(* IEC 61131-3 sources: WATT_Offline/HTB/Prolabs/Alchemy/1. 10.10.110.21/Git, 6 files *)

(* ---- bottle_filling.st ---- *)
PROGRAM botte_filling
  VAR_INPUT
    start : BOOL;
    stop : BOOL;
    overflow_sensor : BOOL;
    filling_sensor : BOOL;
    level_sensor : BOOL;
    capping_sensor : BOOL;
    cap_lazer_sensor : BOOL;
    empty_tank_sensor : BOOL;
  END_VAR
  VAR_OUTPUT
    process_start : BOOL;
    solenoid_valve : BOOL;
    motor_cap : BOOL;
    conveyor_motor : BOOL;
  END_VAR
  VAR
    batch_completed : BOOL;
    sp_beer_flow : INT;
    batch_no : INT;
    current_batch : INT;
    CTU0 : CTU;
    R_TRIG1 : R_TRIG;
  END_VAR

  process_start := NOT(empty_tank_sensor) AND NOT(overflow_sensor) AND NOT(stop) AND (process_start OR start);

  // Hardcoded value min:0 max:100
  sp_beer_flow := 5;

  conveyor_motor := (NOT(motor_cap) OR NOT(capping_sensor)) AND process_start AND (NOT(solenoid_valve) OR NOT(filling_sensor));
  solenoid_valve := NOT(level_sensor) AND (filling_sensor OR solenoid_valve) AND process_start;
  motor_cap := NOT(cap_lazer_sensor) AND (capping_sensor OR motor_cap) AND process_start;
  R_TRIG1(CLK := motor_cap);
  CTU0(CU := R_TRIG1.Q, R := NOT(process_start), PV := batch_no);
  batch_completed := CTU0.Q;
  current_batch := CTU0.CV;
END_PROGRAM

CONFIGURATION Config0

  RESOURCE Res0 ON PLC
    TASK task0(INTERVAL := T#10ms,PRIORITY := 0);
    PROGRAM instance0 WITH task0 : botte_filling;
  END_RESOURCE
END_CONFIGURATION

(* ---- conditioning_aging.st ---- *)
PROGRAM pressure_control
  VAR_EXTERNAL
    master : BOOL;
  END_VAR
  VAR_INPUT
    pressure_sensor : INT := 10;
  END_VAR
  VAR_OUTPUT
    sp_pressure : INT;
    pressure_valve : BOOL;
    open_pressure_valve : BOOL;
    close_pressure_valve : BOOL;
  END_VAR
  VAR
    _TMP_ADD52_OUT : INT;
    _TMP_GT14_OUT : BOOL;
    _TMP_SUB48_OUT : INT;
    _TMP_LT51_OUT : BOOL;
  END_VAR

  pressure_valve := NOT(close_pressure_valve) AND open_pressure_valve AND master;
  _TMP_ADD52_OUT := ADD(sp_pressure, 2);
  _TMP_GT14_OUT := GT(pressure_sensor, _TMP_ADD52_OUT);
  open_pressure_valve := master AND _TMP_GT14_OUT;
  _TMP_SUB48_OUT := SUB(sp_pressure, 2);
  _TMP_LT51_OUT := LT(pressure_sensor, _TMP_SUB48_OUT);
  close_pressure_valve := master AND _TMP_LT51_OUT;
END_PROGRAM

PROGRAM temperature_control
  VAR_EXTERNAL
    master : BOOL;
  END_VAR
  VAR_INPUT
    temp : INT;
  END_VAR
  VAR_OUTPUT
    heater : BOOL;
    sp_heater : INT;
    heater_start : BOOL;
    heater_stop : BOOL;
    cooler : BOOL;
    sp_cooler : INT;
    cooler_start : BOOL;
    cooler_stop : BOOL;
  END_VAR
  VAR
    _TMP_SUB48_OUT : INT;
    _TMP_LT51_OUT : BOOL;
    _TMP_ADD52_OUT : INT;
    _TMP_GT14_OUT : BOOL;
    _TMP_ADD45_OUT : INT;
    _TMP_GT9_OUT : BOOL;
    _TMP_SUB41_OUT : INT;
    _TMP_LT44_OUT : BOOL;
  END_VAR

  heater := NOT(heater_stop) AND (heater OR heater_start) AND master;
  _TMP_SUB48_OUT := SUB(sp_heater, 2);
  _TMP_LT51_OUT := LT(temp, _TMP_SUB48_OUT);
  heater_start := master AND _TMP_LT51_OUT;
  _TMP_ADD52_OUT := ADD(sp_heater, 2);
  _TMP_GT14_OUT := GT(temp, _TMP_ADD52_OUT);
  heater_stop := master AND _TMP_GT14_OUT;
  cooler := NOT(cooler_stop) AND (cooler OR cooler_start) AND master;
  _TMP_ADD45_OUT := ADD(sp_cooler, 2);
  _TMP_GT9_OUT := GT(temp, _TMP_ADD45_OUT);
  cooler_start := master AND _TMP_GT9_OUT;
  _TMP_SUB41_OUT := SUB(sp_cooler, 2);
  _TMP_LT44_OUT := LT(temp, _TMP_SUB41_OUT);
  cooler_stop := master AND _TMP_LT44_OUT;
END_PROGRAM

PROGRAM conditioning
  VAR_EXTERNAL
    master : BOOL;
  END_VAR
  VAR_INPUT
    start : BOOL;
    stop : BOOL;
    open_output_valve : BOOL;
    ultrasonic_level : INT;
  END_VAR
  VAR_OUTPUT
    cycle_on : BOOL;
    intake_pump_material_a : BOOL;
    stop_intake_a : BOOL;
    output_valve : BOOL;
    conditioning_completed : BOOL;
    sp_conditioning_time : INT;
    sp_material_a : INT;
    elapsed_time : INT;
    conditioing_time : TIME;
    elapsed_time_t : TIME;
  END_VAR
  VAR
    TON0 : TON;
    _TMP_GE15_OUT : BOOL;
    _TMP_INT_TO_TIME67_OUT : TIME;
    _TMP_TIME_TO_INT68_OUT : INT;
  END_VAR

  cycle_on := NOT(stop) AND (cycle_on OR start);
  master := NOT(stop) AND (cycle_on OR start);
  intake_pump_material_a := NOT(stop_intake_a) AND cycle_on;
  _TMP_GE15_OUT := GE(ultrasonic_level, sp_material_a);
  stop_intake_a := cycle_on AND _TMP_GE15_OUT;
  _TMP_INT_TO_TIME67_OUT := INT_TO_TIME(sp_conditioning_time);
  conditioing_time := _TMP_INT_TO_TIME67_OUT;
  TON0(IN := stop_intake_a AND cycle_on, PT := conditioing_time);
  conditioning_completed := TON0.Q;
  elapsed_time_t := TON0.ET;
  _TMP_TIME_TO_INT68_OUT := TIME_TO_INT(elapsed_time_t);
  elapsed_time := _TMP_TIME_TO_INT68_OUT;
  output_valve := open_output_valve AND conditioning_completed AND cycle_on;
END_PROGRAM

CONFIGURATION Config0

  RESOURCE Res0 ON PLC
    VAR_GLOBAL
      master : BOOL;
    END_VAR
    TASK task0(INTERVAL := T#1s0ms,PRIORITY := 0);
    TASK task1(INTERVAL := T#1s0ms,PRIORITY := 0);
    TASK task2(INTERVAL := T#1s0ms,PRIORITY := 0);
    PROGRAM instance0 WITH task0 : conditioning;
    PROGRAM instance2 WITH task0 : pressure_control;
    PROGRAM instance1 WITH task1 : temperature_control;
  END_RESOURCE
END_CONFIGURATION

(* ---- fermentation.st ---- *)
PROGRAM fermentation
  VAR_OUTPUT
    sp201 : INT;
    sp202 : INT;
    sp203 : INT;
    sp204 : INT;
  END_VAR
  VAR_EXTERNAL
    MASTER : BOOL;
  END_VAR
  VAR_INPUT
    Start : BOOL;
    Stop : BOOL;
    ultrasonic_level : INT;
  END_VAR
  VAR_OUTPUT
    cycle_on : BOOL;
    intake_pump_material_a : BOOL;
    intake_pump_material_b : BOOL;
    stop_intake_a : BOOL;
    stop_intake_b : BOOL;
    allow_intake_b : BOOL;
    agitator_motor : BOOL;
    stage_timer : BOOL;
    stage_completed : BOOL;
    stage_time : TIME;
    elapsed_stage_timer : TIME;
    elapsed_stage_time : INT;
    sp_agitator_speed : INT;
    next_stage : BOOL;
  END_VAR
  VAR_INPUT
    temp_sensor : INT;
  END_VAR
  VAR_OUTPUT
    stop_agitation : BOOL;
  END_VAR
  VAR
    TON1 : TON;
    _TMP_GE15_OUT : BOOL;
    _TMP_GE9_OUT : BOOL;
    _TMP_GE77_OUT : BOOL;
    _TMP_INT_TO_TIME72_OUT : TIME;
    _TMP_TIME_TO_INT79_OUT : INT;
  END_VAR

  cycle_on := NOT(Stop) AND (Start OR cycle_on);
  MASTER := NOT(Stop) AND (Start OR cycle_on);

  intake_pump_material_a := NOT(stop_intake_a) AND cycle_on;

  _TMP_GE15_OUT := GE(ultrasonic_level, sp201);
  stop_intake_a := cycle_on AND _TMP_GE15_OUT;

  intake_pump_material_b := NOT(stop_intake_b) AND (allow_intake_b OR intake_pump_material_b) AND

  stop_intake_a AND cycle_on;

  _TMP_GE9_OUT := GE(temp_sensor, sp203);
  allow_intake_b := _TMP_GE9_OUT;

  _TMP_GE77_OUT := GE(ultrasonic_level, sp202);
  stop_intake_b := cycle_on AND _TMP_GE77_OUT;

  _TMP_INT_TO_TIME_MIN72_OUT := INT_TO_TIME_MIN(sp204);
  stage_time := _TMP_INT_TO_TIME_MIN72_OUT;

  agitator_motor := NOT(stop_agitation) AND (agitator_motor OR stop_intake_a) AND cycle_on;

  TON1(IN := next_stage AND cycle_on, PT := stage_time);
  stage_timer := TON1.Q;
  elapsed_stage_timer := TON1.ET;

  _TMP_TIME_TO_INT79_OUT := TIME_TO_INT(elapsed_stage_timer);
  elapsed_stage_time := _TMP_TIME_TO_INT79_OUT;

  stage_completed := stage_timer AND cycle_on;
END_PROGRAM

PROGRAM pressure_control
  VAR_EXTERNAL
    MASTER : BOOL;
  END_VAR
  VAR_OUTPUT
    sp208 : INT;
    sp209 : INT;
  END_VAR
  VAR_INPUT
    pressure_sensor : INT;
  END_VAR
  VAR_OUTPUT
    pressure_valve : BOOL;
    open_pressure_valve : BOOL;
    close_pressure_valve : BOOL;
  END_VAR
  VAR
    _TMP_ADD52_OUT : INT;
    _TMP_GT14_OUT : BOOL;
    _TMP_SUB48_OUT : INT;
    _TMP_LT51_OUT : BOOL;
  END_VAR

  pressure_valve := NOT(close_pressure_valve) AND open_pressure_valve AND MASTER;
  _TMP_ADD52_OUT := ADD(sp208, sp209);
  _TMP_GT14_OUT := GT(pressure_sensor, _TMP_ADD52_OUT);
  open_pressure_valve := MASTER AND _TMP_GT14_OUT;
  _TMP_SUB48_OUT := SUB(sp208, sp209);
  _TMP_LT51_OUT := LT(pressure_sensor, _TMP_SUB48_OUT);
  close_pressure_valve := MASTER AND _TMP_LT51_OUT;
END_PROGRAM

PROGRAM pH_control
  VAR_EXTERNAL
    MASTER : BOOL;
  END_VAR
  VAR_OUTPUT
    sp210 : INT;
    sp211 : INT;
    sp212 : INT;
    active : BOOL;
    base_pump : BOOL;
    base_start : BOOL;
    base_stop : BOOL;
    acid_pump : BOOL;
    acid_start : BOOL;
    acid_stop : BOOL;
  END_VAR
  VAR_INPUT
    ph_sensor : INT;
  END_VAR
  VAR
    _TMP_SUB48_OUT : INT;
    _TMP_LT51_OUT : BOOL;
    _TMP_ADD45_OUT : INT;
    _TMP_GT9_OUT : BOOL;
    _TMP_ADD52_OUT : INT;
    _TMP_GT14_OUT : BOOL;
    _TMP_SUB41_OUT : INT;
    _TMP_LT44_OUT : BOOL;
  END_VAR

  base_pump := NOT(base_stop) AND (base_pump OR base_start) AND MASTER;
  acid_pump := NOT(acid_stop) AND (acid_pump OR acid_start) AND MASTER;

  _TMP_SUB48_OUT := SUB(sp210, sp211);
  _TMP_LT51_OUT := LT(ph_sensor, _TMP_SUB48_OUT);
  base_start := MASTER AND _TMP_LT51_OUT;

  _TMP_ADD45_OUT := ADD(sp210, sp212);
  _TMP_GT9_OUT := GT(ph_sensor, _TMP_ADD45_OUT);
  acid_start := MASTER AND _TMP_GT9_OUT;

  _TMP_ADD52_OUT := ADD(sp210, sp211);
  _TMP_GT14_OUT := GT(ph_sensor, _TMP_ADD52_OUT);
  base_stop := MASTER AND _TMP_GT14_OUT;

  _TMP_SUB41_OUT := SUB(sp210, sp212);
  _TMP_LT44_OUT := LT(ph_sensor, _TMP_SUB41_OUT);
  acid_stop := MASTER AND _TMP_LT44_OUT;
END_PROGRAM

PROGRAM temperature_control
  VAR_EXTERNAL
    MASTER : BOOL;
  END_VAR
  VAR_OUTPUT
    sp205 : INT;
    sp206 : INT;
    sp207 : INT;
  END_VAR
  VAR_INPUT
    temp_sensor : INT;
  END_VAR
  VAR_OUTPUT
    heater : BOOL;
    heater_start : BOOL;
    heater_stop : BOOL;
    cooler : BOOL;
    cooler_start : BOOL;
    cooler_stop : BOOL;
  END_VAR
  VAR
    _TMP_SUB48_OUT : INT;
    _TMP_LT51_OUT : BOOL;
    _TMP_ADD45_OUT : INT;
    _TMP_GT9_OUT : BOOL;
    _TMP_ADD52_OUT : INT;
    _TMP_GT14_OUT : BOOL;
    _TMP_SUB41_OUT : INT;
    _TMP_LT44_OUT : BOOL;
  END_VAR

  heater := NOT(heater_stop) AND (heater OR heater_start) AND MASTER;
  cooler := NOT(cooler_stop) AND (cooler OR cooler_start) AND MASTER;

  _TMP_SUB48_OUT := SUB(sp205, sp207);
  _TMP_LT51_OUT := LT(temp_sensor, _TMP_SUB48_OUT);
  heater_start := MASTER AND _TMP_LT51_OUT;

  _TMP_ADD45_OUT := ADD(sp206, sp207);
  _TMP_GT9_OUT := GT(temp_sensor, _TMP_ADD45_OUT);
  cooler_start := MASTER AND _TMP_GT9_OUT;

  _TMP_ADD52_OUT := ADD(sp205, sp207);
  _TMP_GT14_OUT := GT(temp_sensor, _TMP_ADD52_OUT);
  heater_stop := MASTER AND _TMP_GT14_OUT;

  _TMP_SUB41_OUT := SUB(sp206, sp207);
  _TMP_LT44_OUT := LT(temp_sensor, _TMP_SUB41_OUT);
  cooler_stop := MASTER AND _TMP_LT44_OUT;
END_PROGRAM

PROGRAM od_control
  VAR_EXTERNAL
    MASTER : BOOL;
  END_VAR
  VAR_OUTPUT
    sp213 : INT;
    sp214 : INT;
  END_VAR
  VAR_INPUT
    do_sensor : INT;
  END_VAR
  VAR_OUTPUT
    aeration_valve : BOOL;
    open_valve : BOOL;
    close_valve : BOOL;
  END_VAR
  VAR
    _TMP_SUB48_OUT : INT;
    _TMP_LT51_OUT : BOOL;
    _TMP_ADD52_OUT : INT;
    _TMP_GE53_OUT : BOOL;
  END_VAR

  aeration_valve := NOT(close_valve) AND (aeration_valve OR open_valve) AND MASTER;

  _TMP_SUB48_OUT := SUB(sp213, sp214);
  _TMP_LT51_OUT := LT(do_sensor, _TMP_SUB48_OUT);
  open_valve := MASTER AND _TMP_LT51_OUT;

  _TMP_ADD52_OUT := ADD(sp213, sp214);
  _TMP_GE53_OUT := GE(do_sensor, _TMP_ADD52_OUT);
  close_valve := MASTER AND _TMP_GE53_OUT;
END_PROGRAM

CONFIGURATION Config0

  RESOURCE Res0 ON PLC
    VAR_GLOBAL
      MASTER : BOOL;
    END_VAR
    TASK task0(INTERVAL := T#20ms,PRIORITY := 0);
    TASK task1(INTERVAL := T#20ms,PRIORITY := 0);
    TASK task2(INTERVAL := T#20ms,PRIORITY := 0);
    TASK task3(INTERVAL := T#20ms,PRIORITY := 0);
    TASK task4(INTERVAL := T#20ms,PRIORITY := 0);
    PROGRAM instance0 WITH task0 : fermentation;
    PROGRAM instance2 WITH task0 : pressure_control;
    PROGRAM instance4 WITH task0 : od_control;
    PROGRAM instance1 WITH task1 : temperature_control;
    PROGRAM instance3 WITH task3 : pH_control;
  END_RESOURCE
END_CONFIGURATION

(* ---- lautering.st ---- *)
PROGRAM lauter_tun
  VAR_INPUT
    start : BOOL;
    stop : BOOL;
    turbidity_sensor : INT;
    ultra_level_sensor : INT;
  END_VAR
  VAR_OUTPUT
    process_start : BOOL;
    output_valve : BOOL;
    intake_a : BOOL;
    sparge_water_valve : BOOL;
    stop_intake_a : BOOL;
    stop_sparge_water : BOOL;
    rake : BOOL;
    recirculation_pump : BOOL;
    rake_stop : BOOL;
    r_pump_stop : BOOL;
    settling_completed : BOOL;
    grain_removal : BOOL;
    stop_first_runoff : BOOL;
    stop_removal : BOOL;
    stop_final_runoff : BOOL;
    sp_mash_lvl AT %MW10 : INT;
    sp_sparge_water_temp AT %MW11 : INT;
    sp_settle_phase AT %MW51 : INT;
    sp_sparge_water_lvl AT %MW52 : INT;
    sp_first_runoff AT %MW44 : INT;
    sp_grain_bed_level AT %MW35 : INT;
    sp_turbidity_rake AT %MW23 : INT;
    sp_turbidity_vor AT %MW22 : INT;
  END_VAR
  VAR
    settle_phase_pt : TIME;
    settle_phase_et : TIME;
    sp_rake_timer : TIME;
    TON1 : TON;
    TON0 : TON;
    _TMP_GE28_OUT : BOOL;
    _TMP_INT_TO_TIME91_OUT : TIME;
    _TMP_LT62_OUT : BOOL;
    _TMP_LE89_OUT : BOOL;
    _TMP_LE102_OUT : BOOL;
    _TMP_GE107_OUT : BOOL;
    _TMP_LT123_OUT : BOOL;
    _TMP_LT114_OUT : BOOL;
  END_VAR

  process_start := NOT(stop) AND start;
  intake_a := NOT(stop_intake_a) AND process_start;
  _TMP_GE28_OUT := GE(ultra_level_sensor, sp_mash_lvl);
  stop_intake_a := process_start AND _TMP_GE28_OUT OR stop_intake_a AND process_start;
  _TMP_INT_TO_TIME91_OUT := INT_TO_TIME(sp_settle_phase);
  settle_phase_pt := _TMP_INT_TO_TIME91_OUT;
  TON0(IN := stop_intake_a AND process_start, PT := settle_phase_pt);
  settling_completed := TON0.Q;
  settle_phase_et := TON0.ET;
  rake := NOT(rake_stop) AND (rake OR settling_completed) AND process_start;
  _TMP_LT62_OUT := LT(turbidity_sensor, sp_turbidity_rake);
  TON1(IN := stop_intake_a AND process_start AND _TMP_LT62_OUT, PT := sp_rake_timer);
  rake_stop := TON1.Q;
  recirculation_pump := NOT(r_pump_stop) AND (recirculation_pump OR settling_completed) AND process_start;
  _TMP_LE89_OUT := LE(turbidity_sensor, sp_turbidity_vor);
  r_pump_stop := rake_stop AND process_start AND _TMP_LE89_OUT;
  output_valve := NOT(stop_first_runoff) AND (output_valve OR r_pump_stop) AND process_start;
  _TMP_LE102_OUT := LE(ultra_level_sensor, sp_first_runoff);
  stop_first_runoff := r_pump_stop AND process_start AND _TMP_LE102_OUT OR stop_first_runoff AND process_start;
  sparge_water_valve := NOT(stop_sparge_water) AND stop_first_runoff AND process_start;
  _TMP_GE107_OUT := GE(ultra_level_sensor, sp_sparge_water_lvl);
  stop_sparge_water := stop_first_runoff AND process_start AND _TMP_GE107_OUT OR stop_sparge_water;
  output_valve := NOT(stop_final_runoff) AND (output_valve OR stop_sparge_water) AND process_start;
  _TMP_LT123_OUT := LT(ultra_level_sensor, sp_grain_bed_level);
  stop_final_runoff := stop_sparge_water AND process_start AND _TMP_LT123_OUT;
  grain_removal := NOT(stop_removal) AND (grain_removal OR stop_final_runoff) AND process_start;
  _TMP_LT114_OUT := LT(ultra_level_sensor, 5);
  stop_removal := stop_final_runoff AND process_start AND _TMP_LT114_OUT;
END_PROGRAM

CONFIGURATION Config0

  RESOURCE Res0 ON PLC
    TASK task0(INTERVAL := T#1s0ms,PRIORITY := 0);
    PROGRAM instance0 WITH task0 : lauter_tun;
  END_RESOURCE
END_CONFIGURATION

(* ---- mash_mixing.st ---- *)
PROGRAM pressure_control
  VAR_EXTERNAL
    MASTER : BOOL;
  END_VAR
  VAR_INPUT
    pressure_sensor : INT;
  END_VAR
  VAR_OUTPUT
    sp_pressure : INT;
    pressure_valve : BOOL;
    open_pressure_valve : BOOL;
    close_pressure_valve : BOOL;
  END_VAR
  VAR
    _TMP_ADD52_OUT : INT;
    _TMP_GT14_OUT : BOOL;
    _TMP_SUB48_OUT : INT;
    _TMP_LT51_OUT : BOOL;
  END_VAR

  pressure_valve := NOT(close_pressure_valve) AND open_pressure_valve AND MASTER;
  _TMP_ADD52_OUT := ADD(sp_pressure, 2);
  _TMP_GT14_OUT := GT(pressure_sensor, _TMP_ADD52_OUT);
  open_pressure_valve := MASTER AND _TMP_GT14_OUT;
  _TMP_SUB48_OUT := SUB(sp_pressure, 2);
  _TMP_LT51_OUT := LT(pressure_sensor, _TMP_SUB48_OUT);
  close_pressure_valve := MASTER AND _TMP_LT51_OUT;
END_PROGRAM

PROGRAM heating
  VAR_EXTERNAL
    MASTER : BOOL;
  END_VAR
  VAR_INPUT
    temp : INT;
  END_VAR
  VAR_OUTPUT
    heater : BOOL;
    sp_heater : INT := 64;
    heater_start : BOOL;
    heater_stop : BOOL;
    cooler : BOOL;
    sp_cooler : INT := 60;
    cooler_start : BOOL;
    cooler_stop : BOOL;
  END_VAR
  VAR
    _TMP_SUB48_OUT : INT;
    _TMP_LT51_OUT : BOOL;
    _TMP_ADD45_OUT : INT;
    _TMP_GT9_OUT : BOOL;
    _TMP_ADD52_OUT : INT;
    _TMP_GT14_OUT : BOOL;
    _TMP_SUB41_OUT : INT;
    _TMP_LT44_OUT : BOOL;
  END_VAR

  heater := NOT(heater_stop) AND (heater OR heater_start) AND MASTER;
  cooler := NOT(cooler_stop) AND (cooler OR cooler_start) AND MASTER;
  _TMP_SUB48_OUT := SUB(sp_heater, 2);
  _TMP_LT51_OUT := LT(temp, _TMP_SUB48_OUT);
  heater_start := MASTER AND _TMP_LT51_OUT;
  _TMP_ADD45_OUT := ADD(sp_cooler, 2);
  _TMP_GT9_OUT := GT(temp, _TMP_ADD45_OUT);
  cooler_start := MASTER AND _TMP_GT9_OUT;
  _TMP_ADD52_OUT := ADD(sp_heater, 2);
  _TMP_GT14_OUT := GT(temp, _TMP_ADD52_OUT);
  heater_stop := MASTER AND _TMP_GT14_OUT;
  _TMP_SUB41_OUT := SUB(sp_cooler, 2);
  _TMP_LT44_OUT := LT(temp, _TMP_SUB41_OUT);
  cooler_stop := MASTER AND _TMP_LT44_OUT;
END_PROGRAM

PROGRAM MIXER
  VAR_EXTERNAL
    MASTER : BOOL;
  END_VAR
  VAR_INPUT
    Start : BOOL;
    Stop : BOOL;
    ultrasonic_level : INT;
  END_VAR
  VAR_OUTPUT
    cycle_on : BOOL;
    intake_pump_material_a : BOOL;
    intake_pump_material_b : BOOL;
    stop_intake_a : BOOL;
    stop_intake_b : BOOL;
    agitator_motor : BOOL;
    agitator_timer : BOOL;
    output_valve : BOOL;
    ELS : BOOL;
  END_VAR
  VAR
    agitator_time : TIME;
    elapsed_agitation_time : TIME;
  END_VAR
  VAR_OUTPUT
    elapsed_agitation : INT;
    sp_agitator_time : INT;
    sp_agitator_speed : INT;
    sp_material_a : INT;
    sp_material_b : INT;
  END_VAR
  VAR
    TON1 : TON;
    _TMP_INT_TO_TIME72_OUT : TIME;
    _TMP_GE15_OUT : BOOL;
    _TMP_TIME_TO_INT68_OUT : INT;
    _TMP_GE77_OUT : BOOL;
  END_VAR

  cycle_on := NOT(Stop) AND (Start OR cycle_on);
  _TMP_INT_TO_TIME72_OUT := INT_TO_TIME(sp_agitator_time);
  agitator_time := _TMP_INT_TO_TIME72_OUT;
  MASTER := NOT(Stop) AND (Start OR cycle_on)
  agitator_motor := NOT(agitator_timer) AND (agitator_motor OR stop_intake_a) AND cycle_on;
  intake_pump_material_a := NOT(stop_intake_a) AND (intake_pump_material_a AND cycle_on OR cycle_on);
  TON1(IN := stop_intake_b AND cycle_on, PT := agitator_time);
  agitator_timer := TON1.Q;
  elapsed_agitation_time := TON1.ET;
  _TMP_GE15_OUT := GE(ultrasonic_level, sp_material_a);
  stop_intake_a := cycle_on AND _TMP_GE15_OUT;
  _TMP_TIME_TO_INT68_OUT := TIME_TO_INT(elapsed_agitation_time);
  elapsed_agitation := _TMP_TIME_TO_INT68_OUT;
  intake_pump_material_b := NOT(stop_intake_b) AND stop_intake_a AND cycle_on;
  output_valve := NOT(ELS) AND (agitator_timer OR output_valve) AND cycle_on;
  _TMP_GE77_OUT := GE(ultrasonic_level, sp_material_b);
  stop_intake_b := cycle_on AND _TMP_GE77_OUT;
END_PROGRAM

CONFIGURATION Config0

  RESOURCE Res0 ON PLC
    VAR_GLOBAL
      MASTER : BOOL;
    END_VAR
    TASK task0(INTERVAL := T#1s0ms,PRIORITY := 0);
    TASK task1(INTERVAL := T#1s0ms,PRIORITY := 0);
    TASK task2(INTERVAL := T#1s0ms,PRIORITY := 0);
    PROGRAM instance0 WITH task0 : MIXER;
    PROGRAM instance2 WITH task0 : pressure_control;
    PROGRAM instance1 WITH task1 : heating;
  END_RESOURCE
END_CONFIGURATION

(* ---- wort_boiling.st ---- *)
(*
    NOTE 1: The following setpoints are defined for use by third-party components and
    are not directly manipulated by the PLC logic. These values are forwarded
    to external devices, such as dispenser valves, for operational control.
    This approach allows for centralized configuration while leveraging
    specialized control mechanisms provided by the third-party hardware.

    sp_bittering_hops_amount_1
    sp_bittering_hops_amount_2

    sp_flavor_hops_amount_1
    sp_flavor_hops_amount_2

    sp_aroma_hops_amount_1
    sp_aroma_hops_amount_2

    NOTE 2: The setpoints below are crucial for the operation of both the PLC and third-party components.

    sp_boil_time
    sp_final_boil_time
    sp_bittering_hops_time
    sp_flavor_hops_time
    sp_aroma_hops_time

*)

PROGRAM boiling
  VAR_EXTERNAL
    master : BOOL;
    stop_intake_a : BOOL;
    kettle_temp : INT;
  END_VAR
  VAR_INPUT
    ultrasonic_level : INT;
  END_VAR
  VAR_OUTPUT
    boil_time : TIME;
    boil_timer : TIME;
  END_VAR
  VAR_INPUT
    start : BOOL;
    stop : BOOL;
  END_VAR
  VAR_OUTPUT
    cycle_on : BOOL;
    intake_pump_material_a : BOOL;
    agitator_motor : BOOL;
    end_boil : BOOL;
    output_valve : BOOL;
    ELS : BOOL;
    start_boil : BOOL;
    start_bittering_hops AT %QX1.1 : BOOL;
    start_aroma_hops AT %QX1.2 : BOOL;
    start_flavor_hops AT %QX1.3 : BOOL;
    final_boil : BOOL;
    sp_star_boil_timer_temp : INT;
    sp_agitator_speed : INT;
    sp_material_a : INT;
    sp_boil_time AT %MW3 : INT;
    sp_final_boil_time AT %MW4 : INT;
    sp_bittering_hops_time AT %MW5 : INT;
    sp_flavor_hops_time AT %MW6 : INT;
    sp_aroma_hops_time AT %MW7 : INT;
    sp_bittering_hops_amount_1 AT %MW1024 : INT;
    sp_bittering_hops_amount_2 AT %MW1025 : INT;
    sp_flavor_hops_amount_1 AT %MW1026 : INT;
    sp_flavor_hops_amount_2 AT %MW1027 : INT;
    sp_aroma_hops_amount_1 AT %MW1028 : INT;
    sp_aroma_hops_amount_2 AT %MW1029 : INT;
    boil_timer_int : INT;
  END_VAR
  VAR
    TON1 : TON;
    _TMP_INT_TO_TIME72_OUT : TIME;
    _TMP_GE15_OUT : BOOL;
    _TMP_GE14_OUT : BOOL;
    _TMP_TIME_TO_INT75_OUT : INT;
    _TMP_GE23_OUT : BOOL;
    _TMP_GE34_OUT : BOOL;
    _TMP_GE41_OUT : BOOL;
    _TMP_GE70_OUT : BOOL;
  END_VAR

  // Verify stop button is not pressed and start button pressed or cycle already started
  cycle_on := NOT(stop) AND (cycle_on OR start);
  master := NOT(stop) AND (cycle_on OR start);

  // Open intake valve until stop_intake is True
  intake_pump_material_a := NOT(stop_intake_a) AND cycle_on;

  // Stop intake of material a when desired level is reached
  _TMP_GE15_OUT := GE(ultrasonic_level, sp_material_a);
  stop_intake_a := cycle_on AND _TMP_GE15_OUT;

  // Start boiling
  _TMP_GE14_OUT := GE(kettle_temp, sp_star_boil_timer_temp);
  start_boil := cycle_on AND _TMP_GE14_OUT;

  // boil timer to int
  _TMP_TIME_TO_INT75_OUT := TIME_TO_INT(boil_timer);
  boil_timer_int := _TMP_TIME_TO_INT75_OUT;

  // Coil control to signal when to start bittering hops addition
  _TMP_GE23_OUT := GE(boil_timer_int, sp_bittering_hops_time);
  start_bittering_hops := NOT(start_flavor_hops) AND cycle_on AND _TMP_GE23_OUT;

  // Coil control to signal when to start flavor hops addition
  _TMP_GE34_OUT := GE(boil_timer_int, sp_flavor_hops_time);
  start_flavor_hops := NOT(start_aroma_hops) AND cycle_on AND _TMP_GE34_OUT;

  // Coil control to signal when to start aroma hops addition
  _TMP_GE41_OUT := GE(boil_timer_int, sp_aroma_hops_time);
  start_aroma_hops := NOT(final_boil) AND cycle_on AND _TMP_GE41_OUT;

  // Coil to signal final boil started
  _TMP_GE70_OUT := GE(boil_timer_int, sp_final_boil_time);
  final_boil := cycle_on AND _TMP_GE70_OUT;

  // Int to Time boil time
  _TMP_INT_TO_TIME72_OUT := INT_TO_TIME(sp_boil_time);
  boil_time := _TMP_INT_TO_TIME72_OUT;

  // Coil to control agitator motor
  agitator_motor := NOT(end_boil) AND (agitator_motor OR stop_intake_a) AND cycle_on;

  // Coil control to signal end of boiling time
  TON1(IN := start_boil AND cycle_on, PT := boil_time);
  end_boil := TON1.Q;
  boil_timer := TON1.ET;

  // Output valve control
  output_valve := NOT(ELS) AND (end_boil OR output_valve) AND cycle_on;
END_PROGRAM

PROGRAM pressure_control
  VAR_EXTERNAL
    master : BOOL;
  END_VAR
  VAR_INPUT
    pressure_sensor : INT;
  END_VAR
  VAR_OUTPUT
    sp_pressure : INT;
    pressure_valve : BOOL;
    open_pressure_valve : BOOL;
    close_pressure_valve : BOOL;
  END_VAR
  VAR
    _TMP_ADD52_OUT : INT;
    _TMP_GT14_OUT : BOOL;
    _TMP_SUB48_OUT : INT;
    _TMP_LT51_OUT : BOOL;
  END_VAR

  pressure_valve := NOT(close_pressure_valve) AND open_pressure_valve AND master;
  _TMP_ADD52_OUT := ADD(sp_pressure, 2);
  _TMP_GT14_OUT := GT(pressure_sensor, _TMP_ADD52_OUT);
  open_pressure_valve := master AND _TMP_GT14_OUT;
  _TMP_SUB48_OUT := SUB(sp_pressure, 2);
  _TMP_LT51_OUT := LT(pressure_sensor, _TMP_SUB48_OUT);
  close_pressure_valve := master AND _TMP_LT51_OUT;
END_PROGRAM

PROGRAM heating
  VAR_EXTERNAL
    master : BOOL;
    stop_intake_a : BOOL;
    kettle_temp : INT;
  END_VAR
  VAR_INPUT
    temp : INT;
  END_VAR
  VAR_OUTPUT
    heater : BOOL;
    sp_heater : INT;
    heater_start : BOOL;
    heater_stop : BOOL;
    cooler : BOOL;
    sp_cooler : INT;
    cooler_start : BOOL;
    cooler_stop : BOOL;
  END_VAR
  VAR
    _TMP_SUB48_OUT : INT;
    _TMP_LT51_OUT : BOOL;
    _TMP_ADD45_OUT : INT;
    _TMP_GT9_OUT : BOOL;
    _TMP_ADD52_OUT : INT;
    _TMP_GT14_OUT : BOOL;
    _TMP_SUB41_OUT : INT;
    _TMP_LT44_OUT : BOOL;
  END_VAR

  heater := NOT(heater_stop) AND (heater OR heater_start) AND stop_intake_a AND master;
  _TMP_SUB48_OUT := SUB(sp_heater, 2);
  _TMP_LT51_OUT := LT(temp, _TMP_SUB48_OUT);
  heater_start := master AND _TMP_LT51_OUT;
  _TMP_ADD52_OUT := ADD(sp_heater, 2);
  _TMP_GT14_OUT := GT(temp, _TMP_ADD52_OUT);
  heater_stop := master AND _TMP_GT14_OUT;
  kettle_temp := temp;
  cooler := NOT(cooler_stop) AND (cooler OR cooler_start) AND stop_intake_a AND master;
  _TMP_ADD45_OUT := ADD(sp_cooler, 2);
  _TMP_GT9_OUT := GT(temp, _TMP_ADD45_OUT);
  cooler_start := master AND _TMP_GT9_OUT;
  _TMP_SUB41_OUT := SUB(sp_cooler, 2);
  _TMP_LT44_OUT := LT(temp, _TMP_SUB41_OUT);
  cooler_stop := master AND _TMP_LT44_OUT;

END_PROGRAM

CONFIGURATION Config0

  RESOURCE Res0 ON PLC
    VAR_GLOBAL
      master : BOOL;
      stop_intake_a : BOOL;
      kettle_temp : INT;
    END_VAR
    TASK task0(INTERVAL := T#1s0ms,PRIORITY := 0);
    TASK task1(INTERVAL := T#1s0ms,PRIORITY := 0);
    TASK task2(INTERVAL := T#1s0ms,PRIORITY := 0);
    PROGRAM instance0 WITH task0 : boiling;
    PROGRAM instance2 WITH task0 : pressure_control;
    PROGRAM instance1 WITH task1 : heating;
  END_RESOURCE
END_CONFIGURATION
